Staubli VAL3: staubli.pjx

--- staubli.pjx ---
Parameters version=s7.4 stackSize=5000 millimeterUnit=true
Program file=start.pgx
Program file=stop.pgx
Data file=staubli.dtx

--- start.pgx ---
program start()
begin
  do
    for i=0 to 4
      movej(a[i],flange,vit)
    endFor
    movej(s,flange,vitesse)
    movel(w,flange,vitesse)
    waitEndMove()
  until (false)
end
